TYPE ST_System_KKKW_Parameter :
STRUCT
		AutoQuittierung			: BOOL;
END_STRUCT
END_TYPE

(* stored: Version 1.1.0.1, ProductVersion 3.1.4024.9
   DUT ST_System_KKKW_Parameter: Id {d3ec97a4-56fc-4170-acfe-bb57522930e3} *)
